PROGRAM p_EtherCATDiag
VAR
	fbEcatDiag1	:	FB_EcatDiag;
END_VAR

fbEcatDiag1(i_AMSNetId:=g_aEcatMaster1, i_xFirstPass:=g_xFirstPass, q_xAllStatesGood=>g_xIOState);

END_PROGRAM

(* stored: Version 1.1.0.1, ProductVersion 3.1.0.26
   POU p_EtherCATDiag: Id {638320e6-8112-4f35-b44d-c25b584ef133} *)
